(* CODESYS project raduga_prod.project

Project tree, tasks and I/O mapping:
  Device : Owen SPK2xx 03.CS.WEB, Owen, order no. 023, version 3.5.4.20
    application Application
      libraries: Standard, * (System); Util, 3.5.1.0 (System)
      task MainTask (cyclic, interval t#200ms, priority 2) calls PLC_PRG
      task VISU_TASK (cyclic, interval t#200ms, priority 30) calls VisuElems.Visu_Prg
      task AlarmManagerTask (cyclic, interval 50 ms, priority 31) calls AlarmManager.Alarm_Prg
      task bus_task (cyclic, interval t#100ms, priority 1, watchdog t#1000ms x 1) calls MV110
      program PLC_PRG [ST]
      visualisation Visualization
      Alarm Configuration
        alarm class Error (priority 10, acknowledge REP_ACK)
        alarm class Warning (priority 30, acknowledge REP)
        AlarmStorage
        text list AlarmGroup
        alarm group AlarmGroup
            3 [Error]: Comparison Equal, ExpressionToCompare TRUE, Expression PLC_PRG.alm_1 - "Ошибка_1"
            4 [Error]: Comparison Equal, ExpressionToCompare TRUE, Expression PLC_PRG.alm_2 - "Ошибка_2"
            6 [Warning]: Comparison Equal, ExpressionToCompare TRUE, Expression PLC_PRG.accident_sectional_machine - "Авария секционного автомата"
            7 [Warning]: Comparison Equal, ExpressionToCompare TRUE, Expression PLC_PRG.accident_input_1 - "Авария ввода №1"
            44 [Warning]: Comparison Equal, ExpressionToCompare FALSE, Expression PLC_PRG.accident_no_voltage_sec - "Отсутствует напряжение на секции"
            17 [Warning]: Comparison Greater, ExpressionToCompare 32, Expression PLC_PRG.module_in1_Ic - "Перегрузка Ic на вводе №1"
            15 [Warning]: Comparison Greater, ExpressionToCompare 32, Expression PLC_PRG.module_in1_Ia - "Перегрузка Ia на вводе №1"
            25 [Warning]: Comparison Greater, ExpressionToCompare 32, Expression PLC_PRG.module_in2_Ib - "Перегрузка Ib на вводе №2"
            35 [Warning]: Comparison Less, ExpressionToCompare 176, Expression PLC_PRG.module_v1_u3 - "Пониженное напряжение на секции №1 Uc = TRIGGERVALUE"
            13 [Warning]: Comparison Greater, ExpressionToCompare 264, Expression PLC_PRG.module_in1_u3 - "Повышенное напряжение на вводе №1 Uc = TRIGGERVALUE"
            23 [Warning]: Comparison Less, ExpressionToCompare 176, Expression PLC_PRG.module_in2_u3 - "Пониженное напряжение на вводе №2 Uc = TRIGGERVALUE"
            33 [Warning]: Comparison Less, ExpressionToCompare 176, Expression PLC_PRG.module_v1_u2 - "Пониженное напряжение на секции №1 Ub = TRIGGERVALUE"
            43 [Warning]: Comparison Equal, ExpressionToCompare FALSE, Expression PLC_PRG.accident_no_voltage_in_2 - "Отсутствует напряжение на вводе №2"
            21 [Warning]: Comparison Less, ExpressionToCompare 176, Expression PLC_PRG.module_in2_u2 - "Пониженное напряжение на вводе №2 Ub = TRIGGERVALUE"
            31 [Warning]: Comparison Less, ExpressionToCompare 176, Expression PLC_PRG.module_v1_u1 - "Пониженное напряжени на секции №1 Ua = TRIGGERVALUE"
            19 [Warning]: Comparison Less, ExpressionToCompare 176, Expression PLC_PRG.module_in2_u1 - "Пониженное напряжение  на вводе №2 Ua = TRIGGERVALUE"
            16 [Warning]: Comparison Greater, ExpressionToCompare 32, Expression PLC_PRG.module_in1_Ib - "Перегрузка Ib на вводе №1"
            26 [Warning]: Comparison Greater, ExpressionToCompare 32, Expression PLC_PRG.module_in2_Ic - "Перегрузка Ic на вводе №2"
            11 [Warning]: Comparison Greater, ExpressionToCompare 264, Expression PLC_PRG.module_in1_u2 - "Повышенное напряжение на вводе №1 Ub = TRIGGERVALUE"
            14 [Warning]: Comparison Less, ExpressionToCompare 176, Expression PLC_PRG.module_in1_u3 - "Пониженное напряжение Uc на вводе №1 = TRIGGERVALUE"
            24 [Warning]: Comparison Greater, ExpressionToCompare 32, Expression PLC_PRG.module_in2_Ia - "Перегрузка Ia на вводе №2"
            34 [Warning]: Comparison Greater, ExpressionToCompare 264, Expression PLC_PRG.module_v1_u3 - "Повышенное напряжение на секции №1 Uc = TRIGGERVALUE"
            12 [Warning]: Comparison Less, ExpressionToCompare 176, Expression PLC_PRG.module_in1_u2 - "Пониженное напряжение на вводе №1 Ub = TRIGGERVALUE"
            22 [Warning]: Comparison Greater, ExpressionToCompare 264, Expression PLC_PRG.module_in2_u3 - "Повышенное напряжение на вводе №2 Uc = TRIGGERVALUE"
            32 [Warning]: Comparison Greater, ExpressionToCompare 264, Expression PLC_PRG.module_v1_u2 - "Повышенное напряжение на секции №1 Ub = TRIGGERVALUE"
            10 [Warning]: Comparison Less, ExpressionToCompare 176, Expression PLC_PRG.module_in1_u1 - "Пониженное напряжение  на вводе №1 Ua = TRIGGERVALUE"
            20 [Warning]: Comparison Greater, ExpressionToCompare 264, Expression PLC_PRG.module_in2_u2 - "Повышенное напряжение на вводе №2 Ub = TRIGGERVALUE "
            30 [Warning]: Comparison Greater, ExpressionToCompare 264, Expression PLC_PRG.module_v1_u1 - "Повышенное напряжение на секции №1 Ua = TRIGGERVALUE"
            42 [Warning]: Comparison Equal, ExpressionToCompare FALSE, Expression PLC_PRG.accident_no_voltage_in_1 - "Отсутствует напряжение на вводе №1"
            18 [Warning]: Comparison Greater, ExpressionToCompare 264, Expression PLC_PRG.module_in2_u1 - "Повышенное напряжение  на вводе №2 Ua = TRIGGERVALUE"
            8 [Warning]: Comparison Equal, ExpressionToCompare TRUE, Expression PLC_PRG.accident_input_2 - "Авария ввода №2"
            9 [Warning]: Comparison Greater, ExpressionToCompare 264, Expression PLC_PRG.module_in1_u1 - "Повышенное напряжение  на вводе №1 Ua = TRIGGERVALUE"
            0 [Warning]: Comparison Equal, ExpressionToCompare TRUE, Expression PLC_PRG.war_1 - "Предупреждение_1"
            1 [Warning]: Comparison Equal, ExpressionToCompare TRUE, Expression PLC_PRG.war_2 - "Предупреждение_2"
      function block Two_words_to_Real [ST]
      visualisation volt_1
      visualisation mpx_1
      visualisation mpx_2
      visualisation scheme
      image pool ImagePool
    Modbus_COM : Modbus COM, 3S - Smart Software Solutions GmbH, version 3.4.0.0
        settings: DataBits = 8; StopBits = 1; ComPort = 3
      Modbus_Master_COM_Port : Modbus Master, COM Port, 3S - Smart Software Solutions GmbH, version 3.5.5.0
          settings: Transmission = 'RTU'; ResponseTimeout = 1000; TimeBetweenFrames = 10; Auto-restart communication = TRUE
        MV110 : Modbus Slave, COM Port, 3S - Smart Software Solutions GmbH, version 3.5.4.0
            settings: SlaveAddress = 10; ResponseTimeout = 1000; UseExtendedFunctionCodes = TRUE; Channel 0.Function Code = 3; Channel 0.Read Offset = 16#0033; Channel 0.Read Length = 1; Channel 0.Write Offset = 0; Channel 0.Write Length = 0; Channel 0.Cycle Time = 500
            input  Application.PLC_PRG.module_mv110_reg1 : WORD  // Channel 0.Channel 0
            unmapped channels: Channel 0
        MPX_1 : Modbus Slave, COM Port, 3S - Smart Software Solutions GmbH, version 3.5.4.0
            settings: SlaveAddress = 11; ResponseTimeout = 1000; UseExtendedFunctionCodes = TRUE; Input_group.Function Code = 4; Input_group.Read Offset = 16#000B; Input_group.Read Length = 7; Input_group.Write Offset = 0; Input_group.Write Length = 0; Input_group.Cycle Time = 500; Bypass_out_group.Function Code = 3; Bypass_out_group.Read Offset = 16#0015; Bypass_out_group.Read Length = 7; Bypass_out_group.Write Offset = 0; Bypass_out_group.Write Length = 0; Bypass_out_group.Cycle Time = 500; Output_group.Function Code = 3; Output_group.Read Offset = 16#001F; Output_group.Read Length = 13; Output_group.Write Offset = 0; Output_group.Write Length = 0; Output_group.Cycle Time = 500; Battery_group.Function Code = 3; Battery_group.Read Offset = 16#002F; Battery_group.Read Length = 7; Battery_group.Write Offset = 0; Battery_group.Write Length = 0; Battery_group.Cycle Time = 500; temp.Function Code = 3; temp.Read Offset = 16#003D; temp.Read Length = 1; temp.Write Offset = 0; temp.Write Length = 0; temp.Cycle Time = 500; states.Function Code = 3; states.Read Offset = 16#0000; states.Read Length = 2; states.Write Offset = 0; states.Write Length = 0; states.Cycle Time = 500
            input  Application.PLC_PRG.mpx1_in_v_1 : WORD  // Input_group.Input_group
            input  Application.PLC_PRG.mpx1_in_v_2 : WORD  // Input_group.Input_group
            input  Application.PLC_PRG.mpx1_in_v_3 : WORD  // Input_group.Input_group
            input  Application.PLC_PRG.mpx1_in_i_1 : WORD  // Input_group.Input_group
            input  Application.PLC_PRG.mpx1_in_i_2 : WORD  // Input_group.Input_group
            input  Application.PLC_PRG.mpx1_in_i_3 : WORD  // Input_group.Input_group
            input  Application.PLC_PRG.mpx1_in_freq : WORD  // Input_group.Input_group
            input  Application.PLC_PRG.mpx1_bypass_v_1 : WORD  // Bypass_out_group.Bypass_out_group
            input  Application.PLC_PRG.mpx1_bypass_v_2 : WORD  // Bypass_out_group.Bypass_out_group
            input  Application.PLC_PRG.mpx1_bypass_v_3 : WORD  // Bypass_out_group.Bypass_out_group
            input  Application.PLC_PRG.mpx1_bypass_freq : WORD  // Bypass_out_group.Bypass_out_group
            input  Application.PLC_PRG.mpx1_output_v_1 : WORD  // Bypass_out_group.Bypass_out_group
            input  Application.PLC_PRG.mpx1_output_v_2 : WORD  // Bypass_out_group.Bypass_out_group
            input  Application.PLC_PRG.mpx1_output_v_3 : WORD  // Bypass_out_group.Bypass_out_group
            input  Application.PLC_PRG.mpx1_output_i_1 : WORD  // Output_group.Output_group
            input  Application.PLC_PRG.mpx1_output_i_2 : WORD  // Output_group.Output_group
            input  Application.PLC_PRG.mpx1_output_i_3 : WORD  // Output_group.Output_group
            input  Application.PLC_PRG.mpx1_load_ph_1 : WORD  // Output_group.Output_group
            input  Application.PLC_PRG.mpx1_load_ph_2 : WORD  // Output_group.Output_group
            input  Application.PLC_PRG.mpx1_load_ph_3 : WORD  // Output_group.Output_group
            input  Application.PLC_PRG.mpx1_output_active_power_1 : WORD  // Output_group.Output_group
            input  Application.PLC_PRG.mpx1_output_active_power_2 : WORD  // Output_group.Output_group
            input  Application.PLC_PRG.mpx1_output_active_power_3 : WORD  // Output_group.Output_group
            input  Application.PLC_PRG.mpx1_output_freq : WORD  // Output_group.Output_group
            input  Application.PLC_PRG.mpx1_battery_voltage : WORD  // Battery_group.Battery_group
            input  Application.PLC_PRG.mpx1_battery_current : WORD  // Battery_group.Battery_group
            input  Application.PLC_PRG.mpx1_battery_capacity : WORD  // Battery_group.Battery_group
            input  Application.PLC_PRG.mpx1_battery_time : WORD  // Battery_group.Battery_group
            input  Application.PLC_PRG.mpx1_temp : WORD  // temp.temp
            input  Application.PLC_PRG.mpx1_state_reg_1 : WORD  // states.states
            input  Application.PLC_PRG.mpx1_state_reg_2 : WORD  // states.states
            unmapped channels: Input_group, Bypass_out_group, Output_group, Battery_group, temp, states
    Modbus_slave : Modbus COM, 3S - Smart Software Solutions GmbH, version 3.4.0.0
        settings: DataBits = 8; StopBits = 1; ComPort = 4
      Modbus_Serial_Device : Modbus Serial Device, 3S - Smart Software Solutions GmbH, version 3.5.3.80
          settings: Unit-ID = 3
          unmapped channels: Inputs, Outputs
    Ethernet : Ethernet, 3S - Smart Software Solutions GmbH, version 3.4.2.0
      Modbus_TCP_Master : Modbus TCP Master, 3S - Smart Software Solutions GmbH, version 3.5.4.0
          settings: AutoReconnect = TRUE
        IPS_1 : Modbus TCP Slave, 3S - Smart Software Solutions GmbH, version 3.5.4.0
            settings: Unit-ID = 1; ResponseTimeout = 1500; IPAddress = [192, 168, 19, 34]; Input_group.Function Code = 3; Input_group.Read Offset = 16#006E; Input_group.Read Length = 3; Input_group.Write Offset = 0; Input_group.Write Length = 0; Input_group.Cycle Time = 500; Output_group.Function Code = 3; Output_group.Read Offset = 16#0077; Output_group.Read Length = 7; Output_group.Write Offset = 0; Output_group.Write Length = 0; Output_group.Cycle Time = 500; Bypass_group.Function Code = 3; Bypass_group.Read Offset = 16#0081; Bypass_group.Read Length = 4; Bypass_group.Write Offset = 0; Bypass_group.Write Length = 0; Bypass_group.Cycle Time = 500
            unmapped channels: Input_group, Output_group, Bypass_group
    Modbus_PLC_slave : Modbus COM, 3S - Smart Software Solutions GmbH, version 3.4.0.0
        settings: DataBits = 8; StopBits = 1; ComPort = 2
      Modbus_Serial_Device_1 : Modbus Serial Device, 3S - Smart Software Solutions GmbH, version 3.5.5.0
          unmapped channels: Inputs, Outputs
  text list GlobalTextList
  5ce3da45-db07-42e7-a21c-a00fff4ed8f6|D:\scheme_3.png
  5ce3da45-db07-42e7-a21c-a00fff4ed8f6|D:\scheme.png
  5ce3da45-db07-42e7-a21c-a00fff4ed8f6|D:\on.png
  5ce3da45-db07-42e7-a21c-a00fff4ed8f6|D:\off.png
  5ce3da45-db07-42e7-a21c-a00fff4ed8f6|D:\off.jpg
  5ce3da45-db07-42e7-a21c-a00fff4ed8f6|D:\on.jpg
  5ce3da45-db07-42e7-a21c-a00fff4ed8f6|D:\on_ind.jpg
  5ce3da45-db07-42e7-a21c-a00fff4ed8f6|D:\off_ind.jpg
  5ce3da45-db07-42e7-a21c-a00fff4ed8f6|D:\entel.png
  5ce3da45-db07-42e7-a21c-a00fff4ed8f6|D:\zit.png
  5ce3da45-db07-42e7-a21c-a00fff4ed8f6|D:\entel.jpg
  5ce3da45-db07-42e7-a21c-a00fff4ed8f6|D:\zit.jpg
  5ce3da45-db07-42e7-a21c-a00fff4ed8f6|D:\vvod_off.png
  5ce3da45-db07-42e7-a21c-a00fff4ed8f6|D:\vvod_on.png
*)

// Device/Application/PLC_PRG
PROGRAM PLC_PRG
VAR
	alm_1: BOOL;
	alm_2: BOOL;
	war_1: BOOL;
	war_2: BOOL;
	//Переменные для отработки аварийных ситуаций
	accident_sectional_machine :BOOL := FALSE; //авария секционного автомата
	accident_input_1		   :BOOL := FALSE; //авария ввода №1
	accident_input_2		   :BOOL := FALSE; //авария ввода №2
	accident_no_voltage_in_1   :BOOL := FALSE; //отсутствие напряжения на вводе №1
	accident_no_voltage_in_2   :BOOL := FALSE; //отсутствие напряжения на вводе №2
	manual_mode				   :BOOL := FALSE;
	auto_mode                  :BOOL := FALSE;
	remote_mode                :BOOL := FALSE;
	accident_no_voltage_sec    :BOOL := FALSE; //отсутствие напряжения на секции
	
	ack:BOOL;
	history:BOOL;
	
	//Переменные для работы с MPX_1
	mpx1_in_v_1 	 		:WORD; //1-е Напрядение входа
	mpx1_in_v_2 	 :WORD; //2-e Напряжение входа
	mpx1_in_v_3 	 :WORD; //3-е Напряжение входа
	mpx1_in_i_1 	 :WORD; //1-й Ток входа
	mpx1_in_i_2 	 :WORD; //2-й Ток входа
	mpx1_in_i_3 	 :WORD; //3-й Ток входа
	mpx1_in_freq 	 :WORD; //Частота на входе
	mpx1_bypass_v_1  :WORD; //1-е Напряжение байпаса
	mpx1_bypass_v_2  :WORD; //2-е Напряжение байпаса
	mpx1_bypass_v_3  :WORD; //3-е Напряжение байпаса
	mpx1_bypass_freq :WORD; //Частота байпаса
	mpx1_output_v_1  :WORD; //1-е Напряжение выхода
	mpx1_output_v_2  :WORD; //2-е Напряжение выхода
	mpx1_output_v_3  :WORD; //3-е Напряжение выхода
	mpx1_output_i_1  :WORD; //1-й Ток выхода
	mpx1_output_i_2  		   :WORD; //2-й Ток выхода
	mpx1_output_i_3  		   :WORD; //3-й Ток выхода
	mpx1_output_active_power_1 :WORD; //Активная мощность 1-й фазы
	mpx1_output_active_power_2 :WORD; //Активная мощность 2-й фазы
	mpx1_output_active_power_3 :WORD; //Активная мощность 3-й фазы
	mpx1_output_freq :WORD; //Частота выхода
	mpx1_load_ph_1    :WORD; //Загрузска 1-й фазы (%)
	mpx1_load_ph_2    :WORD; //Загрузска 3-й фазы (%)
	mpx1_load_ph_3    :WORD; //Загрузска 2-й фазы (%)
	mpx1_battery_voltage :WORD; //Напряжение батареи
	mpx1_battery_current :WORD; //Ток батареи
	mpx1_battery_capacity :WORD; //Остаточная емкость батареи (%)
	mpx1_battery_time :WORD; //Остаточное время автономии (минуты)
	mpx1_temp :WORD; //Температура
	mpx1_state_reg_1 :WORD; //1-й Регистр состояния
	mpx1_state_1_as_bit :WORD_AS_BIT;
	mpx1_state_reg_2 :WORD; //2-й Регистр состояния
	mpx1_state_2_as_bit :WORD_AS_BIT;
	
	
	
	//Переменные для работы с первым МВ110-16 (адрес = 1)
	module_mv110_reg1	:WORD; //Первый регистр состояния входов МВ110-16
	mv110_reg_as_bit 	:WORD_AS_BIT; 
	mv110_in_1 			:STRING; //РКН ввода 1
	mv110_in_2 			:STRING; //РКН ввода 2
	mv110_in_3 			:STRING; //Сборная шина 1
	mv110_in_4 			:STRING; //Сборная шина 2
	mv110_in_5 			:STRING; //Авария секционного автомата
	mv110_in_6 			:STRING; //Авария ввода 1
	mv110_in_7 			:STRING; //Авария ввода 2
	mv110_in_9 			:STRING; //Положение секционного авт.
	mv110_in_10			:STRING; //Положение ввода 1 авт.
	mv110_in_11			:STRING; //Положение ввода 2 авт.
	mode                :WSTRING := "Старт"; //Режим работы (ручной, ручной дистанционный, автоматический)
	
	
	//Переменные для работы с первым вольтметром (адрес = 3)
	module_v1_u1		:REAL; //Значение Ua первого вольтметра
	module_v1_u2		:REAL; //Значение Ub первого вольтметра
	module_v1_u3		:REAL; //Значение Uc первого вольтметра	
	module_v1_u1_reg1	:WORD; //Первый регистр Ua первого вольтметра
	module_v1_u1_reg2	:WORD; //Второй регистр Ua первого вольтметра
	module_v1_u2_reg1	:WORD; //Первый регистр Ub первого вольтметра
	module_v1_u2_reg2	:WORD; //Второй регистр Ub первого вольтметра
	module_v1_u3_reg1	:WORD; //Первый регистр Uс первого вольтметра
	module_v1_u3_reg2	:WORD; //Второй регистр Uс первого вольтметра		
	module_v1_u1_convertion: Two_words_to_Real;
	module_v1_u2_convertion: Two_words_to_Real;
	module_v1_u3_convertion: Two_words_to_Real;	
	module_v1_F			:REAL; //Значение частоты первого вольтметра	
	module_v1_F_reg1	:WORD; //Первый регистр F первого вольтметра
	module_v1_F_reg2	:WORD; //Второй регистр F первого вольтметра	
	module_v1_F_convertion: Two_words_to_Real;
		
	//Переменные для работы с первым вводом (адрес = 5)
	module_in1_u1		:REAL; //Значение Ua первого ввода
	module_in1_u2		:REAL; //Значение Ub первого ввода
	module_in1_u3		:REAL; //Значение Uc первого ввода	
	module_in1_u1_reg1	:WORD; //Первый регистр Ua первого ввода
	module_in1_u1_reg2	:WORD; //Второй регистр Ua первого ввода
	module_in1_u2_reg1	:WORD; //Первый регистр Ub первого ввода
	module_in1_u2_reg2	:WORD; //Второй регистр Ub первого ввода
	module_in1_u3_reg1	:WORD; //Первый регистр Uс первого ввода
	module_in1_u3_reg2	:WORD; //Второй регистр Uс первого ввода		
	module_in1_u1_convertion: Two_words_to_Real;
	module_in1_u2_convertion: Two_words_to_Real;
	module_in1_u3_convertion: Two_words_to_Real;
	
	module_in1_Uab		:REAL; //Значение Uab первого ввода
	module_in1_Ubc		:REAL; //Значение Ubc первого ввода
	module_in1_Uca		:REAL; //Значение Uca первого ввода	
	module_in1_Uab_reg1	:WORD; //Первый регистр Uab первого ввода
	module_in1_Uab_reg2	:WORD; //Второй регистр Uab первого ввода
	module_in1_Ubc_reg1	:WORD; //Первый регистр Ubc первого ввода
	module_in1_Ubc_reg2	:WORD; //Второй регистр Ubc первого ввода
	module_in1_Uca_reg1	:WORD; //Первый регистр Uсa первого ввода
	module_in1_Uca_reg2	:WORD; //Второй регистр Uсa первого ввода	
	module_in1_Uab_convertion: Two_words_to_Real;
	module_in1_Ubc_convertion: Two_words_to_Real;
	module_in1_Uca_convertion: Two_words_to_Real;
	
	module_in1_Ia		:REAL; //Значение Ia первого ввода
	module_in1_Ib		:REAL; //Значение Ib первого ввода
	module_in1_Ic		:REAL; //Значение Ic первого ввода	
	module_in1_Ia_reg1	:WORD; //Первый регистр Ia первого ввода
	module_in1_Ia_reg2	:WORD; //Второй регистр Ia первого ввода
	module_in1_Ib_reg1	:WORD; //Первый регистр Ib первого ввода
	module_in1_Ib_reg2	:WORD; //Второй регистр Ib первого ввода
	module_in1_Ic_reg1	:WORD; //Первый регистр Iс первого ввода
	module_in1_Ic_reg2	:WORD; //Второй регистр Iс первого ввода	
	module_in1_Ia_convertion: Two_words_to_Real;
	module_in1_Ib_convertion: Two_words_to_Real;
	module_in1_Ic_convertion: Two_words_to_Real;

	module_in1_F		:REAL; //Значение частоты первого ввода
	module_in1_F_reg1	:WORD; //Первый регистр F первого ввода
	module_in1_F_reg2	:WORD; //Второй регистр F первого ввода	
	module_in1_F_convertion: Two_words_to_Real;
	
	//Переменные для работы со вторым вводом (адрес = 6)
	module_in2_u1		:REAL; //Значение Ua первого второго
	module_in2_u2		:REAL; //Значение Ub первого второго
	module_in2_u3		:REAL; //Значение Uc первого второго	
	module_in2_u1_reg1	:WORD; //Первый регистр Ua первого второго
	module_in2_u1_reg2	:WORD; //Второй регистр Ua первого второго
	module_in2_u2_reg1	:WORD; //Первый регистр Ub первого второго
	module_in2_u2_reg2	:WORD; //Второй регистр Ub первого второго
	module_in2_u3_reg1	:WORD; //Первый регистр Uс первого второго
	module_in2_u3_reg2	:WORD; //Второй регистр Uс первого второго		
	module_in2_u1_convertion: Two_words_to_Real;
	module_in2_u2_convertion: Two_words_to_Real;
	module_in2_u3_convertion: Two_words_to_Real;
	
	module_in2_Uab		:REAL; //Значение Uab первого ввода
	module_in2_Ubc		:REAL; //Значение Ubc первого ввода
	module_in2_Uca		:REAL; //Значение Uca первого ввода	
	module_in2_Uab_reg1	:WORD; //Первый регистр Uab первого ввода
	module_in2_Uab_reg2	:WORD; //Второй регистр Uab первого ввода
	module_in2_Ubc_reg1	:WORD; //Первый регистр Ubc первого ввода
	module_in2_Ubc_reg2	:WORD; //Второй регистр Ubc первого ввода
	module_in2_Uca_reg1	:WORD; //Первый регистр Uсa первого ввода
	module_in2_Uca_reg2	:WORD; //Второй регистр Uсa первого ввода	
	module_in2_Uab_convertion: Two_words_to_Real;
	module_in2_Ubc_convertion: Two_words_to_Real;
	module_in2_Uca_convertion: Two_words_to_Real;

	module_in2_Ia		:REAL; //Значение Ia первого ввода
	module_in2_Ib		:REAL; //Значение Ib первого ввода
	module_in2_Ic		:REAL; //Значение Ic первого ввода	
	module_in2_Ia_reg1	:WORD; //Первый регистр Ia первого ввода
	module_in2_Ia_reg2	:WORD; //Второй регистр Ia первого ввода
	module_in2_Ib_reg1	:WORD; //Первый регистр Ib первого ввода
	module_in2_Ib_reg2	:WORD; //Второй регистр Ib первого ввода
	module_in2_Ic_reg1	:WORD; //Первый регистр Iс первого ввода
	module_in2_Ic_reg2	:WORD; //Второй регистр Iс первого ввода	
	module_in2_Ia_convertion: Two_words_to_Real;
	module_in2_Ib_convertion: Two_words_to_Real;
	module_in2_Ic_convertion: Two_words_to_Real;
	
	module_in2_F		:REAL; //Значение частоты первого ввода
	module_in2_F_reg1	:WORD; //Первый регистр F первого ввода
	module_in2_F_reg2	:WORD; //Второй регистр F первого ввода	
	module_in2_F_convertion: Two_words_to_Real;
END_VAR

//Конвертация параметров mpx_1




//Конвертация 2 считанных регистров типа WORD в одну переменную REAL для каждого измеряемого значения
//Первый вольтметр (адрес = 3)
module_v1_u1_convertion(Inpit_1:=module_v1_u1_reg1 , Inpit_2:=module_v1_u1_reg2 , output=>module_v1_u1 ); //V1 Ua
module_v1_u2_convertion(Inpit_1:=module_v1_u2_reg1 , Inpit_2:=module_v1_u2_reg2 , output=>module_v1_u2 ); //V1 Ub
module_v1_u3_convertion(Inpit_1:=module_v1_u3_reg1 , Inpit_2:=module_v1_u3_reg2 , output=>module_v1_u3 ); //V1 Uc
module_v1_F_convertion  (Inpit_1:=module_v1_F_reg1,    Inpit_2 := module_v1_F_reg2,   output=>module_v1_F );   //V1 F

//МФИ ввод №1 (адрес = 5)
module_in1_u1_convertion(Inpit_1:=module_in1_u1_reg1 , Inpit_2:=module_in1_u1_reg2 , output=>module_in1_u1 ); //Ua
module_in1_u2_convertion(Inpit_1:=module_in1_u2_reg1 , Inpit_2:=module_in1_u2_reg2 , output=>module_in1_u2 ); //Ub
module_in1_u3_convertion(Inpit_1:=module_in1_u3_reg1 , Inpit_2:=module_in1_u3_reg2 , output=>module_in1_u3 ); //Uc
module_in1_Uab_convertion(Inpit_1:=module_in1_Uab_reg1,  Inpit_2 := module_in1_Uab_reg2, output=>module_in1_Uab ); //Uab
module_in1_Ubc_convertion(Inpit_1:=module_in1_Ubc_reg1,  Inpit_2 := module_in1_Ubc_reg2, output=>module_in1_Ubc ); //Ubc
module_in1_Uca_convertion(Inpit_1:=module_in1_Uca_reg1,  Inpit_2 := module_in1_Uca_reg2, output=>module_in1_Uca ); //Uca
module_in1_F_convertion  (Inpit_1:=module_in1_F_reg1,    Inpit_2 := module_in1_F_reg2,   output=>module_in1_F );//F
module_in1_Ia_convertion  (Inpit_1:=module_in1_Ia_reg1,    Inpit_2 := module_in1_Ia_reg2,   output=>module_in1_Ia );//Ia
module_in1_Ib_convertion  (Inpit_1:=module_in1_Ib_reg1,    Inpit_2 := module_in1_Ib_reg2,   output=>module_in1_Ib );//Ib
module_in1_Ic_convertion  (Inpit_1:=module_in1_Ic_reg1,    Inpit_2 := module_in1_Ic_reg2,   output=>module_in1_Ic );//Ic

//МФИ ввод №2 (адрес = 6)
module_in2_u1_convertion(Inpit_1:=module_in2_u1_reg1 , Inpit_2:=module_in2_u1_reg2 , output=>module_in2_u1 ); //Ua
module_in2_u2_convertion(Inpit_1:=module_in2_u2_reg1 , Inpit_2:=module_in2_u2_reg2 , output=>module_in2_u2 ); //Ub
module_in2_u3_convertion(Inpit_1:=module_in2_u3_reg1 , Inpit_2:=module_in2_u3_reg2 , output=>module_in2_u3 ); //Uc
module_in2_Uab_convertion(Inpit_1:=module_in2_Uab_reg1,  Inpit_2 := module_in2_Uab_reg2, output=>module_in2_Uab ); //Uab
module_in2_Ubc_convertion(Inpit_1:=module_in2_Ubc_reg1,  Inpit_2 := module_in2_Ubc_reg2, output=>module_in2_Ubc ); //Ubc
module_in2_Uca_convertion(Inpit_1:=module_in2_Uca_reg1,  Inpit_2 := module_in2_Uca_reg2, output=>module_in2_Uca ); //Uca
module_in2_F_convertion  (Inpit_1:=module_in2_F_reg1,    Inpit_2 := module_in2_F_reg2,   output=>module_in2_F );//F
module_in2_Ia_convertion  (Inpit_1:=module_in2_Ia_reg1,    Inpit_2 := module_in2_Ia_reg2,   output=>module_in2_Ia );//Ia
module_in2_Ib_convertion  (Inpit_1:=module_in2_Ib_reg1,    Inpit_2 := module_in2_Ib_reg2,   output=>module_in2_Ib );//Ib
module_in2_Ic_convertion  (Inpit_1:=module_in2_Ic_reg1,    Inpit_2 := module_in2_Ic_reg2,   output=>module_in2_Ic );//Ic

//Логика МВ110-16
mv110_reg_as_bit(W := module_mv110_reg1);

IF (mv110_reg_as_bit.B00 = FALSE) THEN
	mv110_in_1 := 'on_ind';
	ELSE
		mv110_in_1 := 'off_ind';	
END_IF
IF (mv110_reg_as_bit.B01 = FALSE) THEN
	mv110_in_2 := 'on_ind';
	ELSE
		mv110_in_2 := 'off_ind';	 
END_IF
IF (mv110_reg_as_bit.B02 = FALSE) THEN
	mv110_in_3 := 'on_ind';
	ELSE
		mv110_in_3 := 'off_ind';	 
END_IF
IF (mv110_reg_as_bit.B03 = FALSE) THEN
	mv110_in_4 := 'on_ind';
	ELSE
		mv110_in_4 := 'off_ind';	 
END_IF
IF (mv110_reg_as_bit.B08 = TRUE) THEN
	mv110_in_9 := 'on';
	ELSE
		mv110_in_9 := 'off';	 
END_IF
IF (mv110_reg_as_bit.B09 = TRUE) THEN
	mv110_in_10 := 'on';
	ELSE
		mv110_in_10 := 'off';	 
END_IF
IF (mv110_reg_as_bit.B10 = TRUE) THEN
	mv110_in_11 := 'on';
	ELSE
		mv110_in_11 := 'off';	 	 
END_IF
IF (mv110_reg_as_bit.B04 = TRUE) THEN
	accident_sectional_machine := TRUE;
	ELSE
		accident_sectional_machine := FALSE;	 	 
END_IF
IF (mv110_reg_as_bit.B05 = TRUE) THEN
	accident_input_1 := TRUE;
	ELSE
		accident_input_1 := FALSE;	 	 
END_IF
IF (mv110_reg_as_bit.B06 = TRUE) THEN
	accident_input_2 := TRUE;
	ELSE
		accident_input_2 := FALSE;	 	 
END_IF
IF (mv110_reg_as_bit.B00 = FALSE) THEN
	accident_no_voltage_in_1 := FALSE;
	ELSE
		accident_no_voltage_in_1 := TRUE;	
END_IF
IF (mv110_reg_as_bit.B01 = FALSE) THEN
	accident_no_voltage_in_2 := FALSE;
	ELSE
		accident_no_voltage_in_2 := TRUE;	 
END_IF
IF (mv110_reg_as_bit.B02 = FALSE) THEN
	accident_no_voltage_sec := FALSE;
	ELSE
		accident_no_voltage_sec := TRUE;	 
END_IF
IF (mv110_reg_as_bit.B12 = TRUE) THEN
	mode := "Автоматический";
	auto_mode := TRUE;
	manual_mode := FALSE;
	remote_mode := FALSE;
END_IF
IF ((mv110_reg_as_bit.B12 = FALSE) AND (mv110_reg_as_bit.B13 = FALSE)) THEN
	mode := "Ручной";
	auto_mode := FALSE;
	manual_mode := TRUE;
	remote_mode := FALSE;
END_IF
IF ((mv110_reg_as_bit.B12 = FALSE) AND (mv110_reg_as_bit.B13 = TRUE)) THEN
	mode := "Дистанционный";
	auto_mode := FALSE;
	manual_mode := FALSE;
	remote_mode := TRUE;
END_IF
//--------------------------


(*открыли порт 3. я откатил до старых версий порты , компилируется.
добавил чтение раз в 100 мс регистра 2и 3 в канале нуль
в закладке соотнесение указал включено 2 = для обновления данных в СПК циклично
склейл два ворда в реал в первой строке этого кода
далее код переподъём  ,в случае  ,если модуль упал ( убрали или ошибки)*)

END_PROGRAM

// Device/Application/Two_words_to_Real
FUNCTION_BLOCK Two_words_to_Real
VAR_INPUT
	Inpit_1:WORD;
	Inpit_2:WORD;
END_VAR
VAR_OUTPUT
	output:real;
END_VAR
VAR
	P:POINTER TO ARRAY [0..3] OF BYTE; 
	pi1:POINTER TO ARRAY [0..1] OF BYTE; 
	pi2:POINTER TO ARRAY [0..1] OF BYTE; 
END_VAR

pi1:=ADR(Inpit_1);
pi2:=ADR(Inpit_2);



P:=ADR(output);
P^[0]:=pi2^[0];
P^[1]:=pi2^[1];
P^[2]:=pi1^[0];
P^[3]:=pi1^[1];

END_FUNCTION_BLOCK

// Device/Application/Visualization
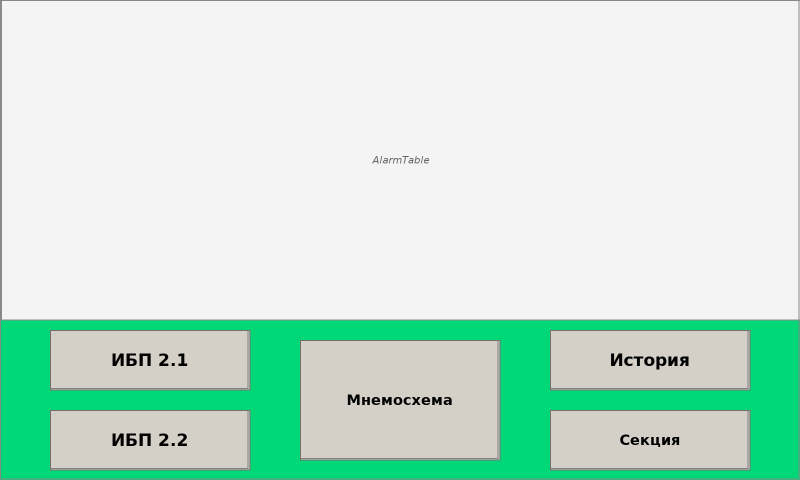
VISUALIZATION Visualization  // 800x480
    AlarmTable (1,0 800x320)
        Column[0]: ColumnTitle=Время
        Column[1]: ColumnTitle=Сообщение
        p1521930926: __All
        p1663851261: __All
        p428520879: PLC_PRG.ack
        p3266827225: PLC_PRG.history
    Button (550,330 200x60), "История", colour toggle: PLC_PRG.history
        toggle PLC_PRG.history
    Button (550,410 200x60), "Секция"
        OnMouseClick:  Assign=volt_1, Type=Assignment
    Button (50,330 200x60), "ИБП 2.1"
        OnMouseClick:  Assign=mpx_1, Type=Assignment
    Button (50,410 200x60), "ИБП 2.2"
        OnMouseClick:  Assign=mpx_2, Type=Assignment
    Button (300,340 200x120), "Мнемосхема"
        OnMouseClick:  Assign=scheme, Type=Assignment
END_VISUALIZATION

// Device/Application/volt_1
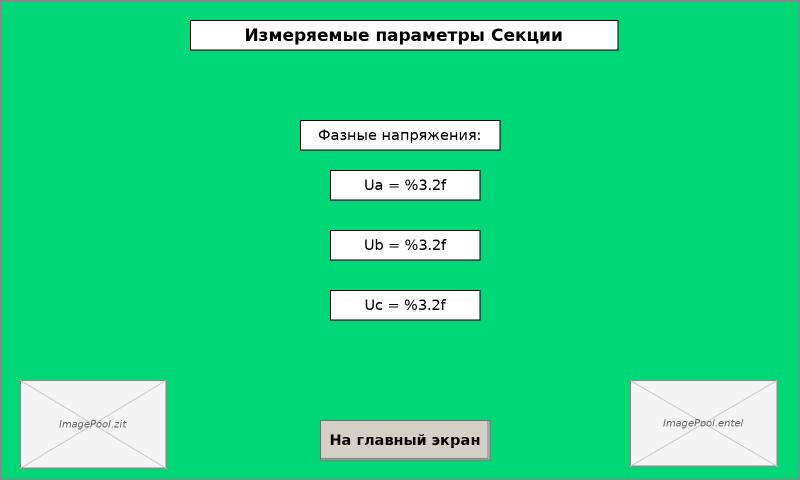
VISUALIZATION volt_1  // 800x480
    Rectangle (190,20 428x30), "Измеряемые параметры Секции"
    Button (320,420 170x40), "На главный экран"
        OnMouseClick:  Assign=Visualization, Type=Assignment
    Rectangle (300,120 200x30), "Фазные напряжения:"
    Rectangle (330,170 150x30), "Ua = %3.2f", text variable: PLC_PRG.module_v1_u1
    Rectangle (330,230 150x30), "Ub = %3.2f", text variable: PLC_PRG.module_v1_u2
    Rectangle (330,290 150x30), "Uc = %3.2f", text variable: PLC_PRG.module_v1_u3
    Image (630,380 147x86), image: ImagePool.entel
    Image (20,380 146x88), image: ImagePool.zit
END_VISUALIZATION

// Device/Application/mpx_1
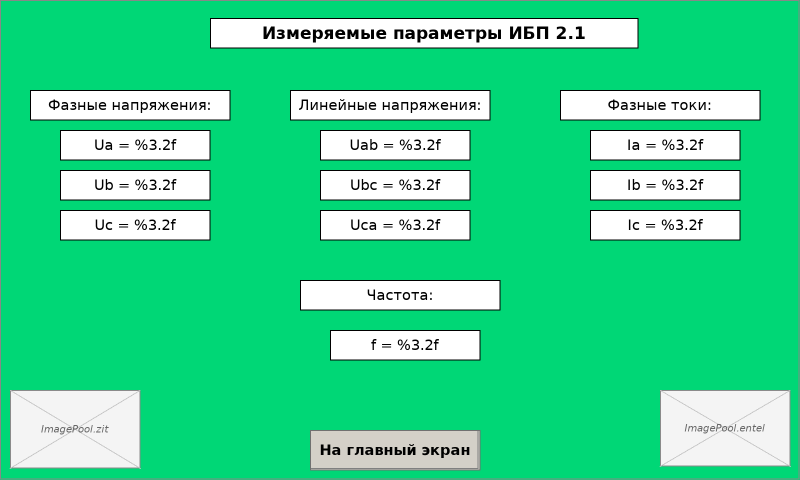
VISUALIZATION mpx_1  // 800x480
    Button (310,430 170x40), "На главный экран"
        OnMouseClick:  Assign=Visualization, Type=Assignment
    Rectangle (210,18 428x30), "Измеряемые параметры ИБП 2.1"
    Rectangle (30,90 200x30), "Фазные напряжения:"
    Rectangle (60,130 150x30), "Ua = %3.2f", text variable: PLC_PRG.module_in1_u1
    Rectangle (60,170 150x30), "Ub = %3.2f", text variable: PLC_PRG.module_in1_u2
    Rectangle (60,210 150x30), "Uc = %3.2f", text variable: PLC_PRG.module_in1_u3
    Rectangle (290,90 200x30), "Линейные напряжения:"
    Rectangle (320,130 150x30), "Uab = %3.2f", text variable: PLC_PRG.module_in1_Uab
    Rectangle (320,170 150x30), "Ubc = %3.2f", text variable: PLC_PRG.module_in1_Ubc
    Rectangle (320,210 150x30), "Uca = %3.2f", text variable: PLC_PRG.module_in1_Uca
    Rectangle (560,90 200x30), "Фазные токи:"
    Rectangle (590,130 150x30), "Ia = %3.2f", text variable: PLC_PRG.module_in1_Ia
    Rectangle (590,170 150x30), "Ib = %3.2f", text variable: PLC_PRG.module_in1_Ib
    Rectangle (590,210 150x30), "Ic = %3.2f", text variable: PLC_PRG.module_in1_Ic
    Rectangle (300,280 200x30), "Частота:"
    Rectangle (330,330 150x30), "f = %3.2f", text variable: PLC_PRG.module_in1_F
    Image (10,390 130x78), image: ImagePool.zit
    Image (660,390 130x76), image: ImagePool.entel
END_VISUALIZATION

// Device/Application/mpx_2
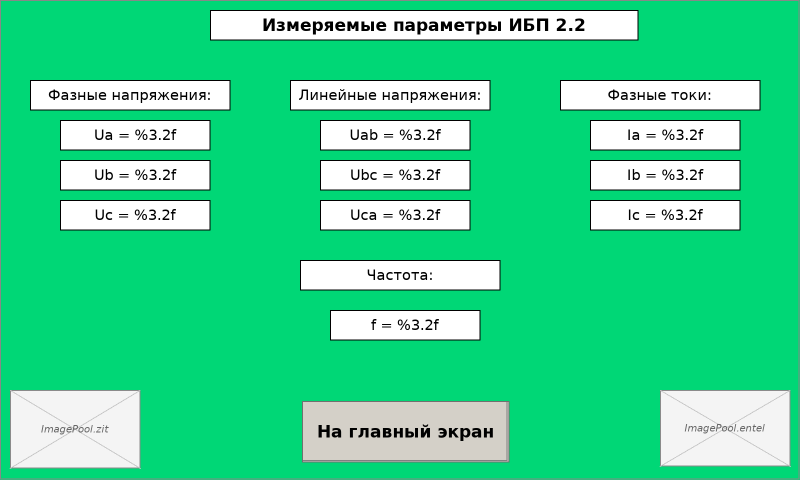
VISUALIZATION mpx_2  // 800x480
    Button (302,401 207x61), "На главный экран"
        OnMouseClick:  Assign=Visualization, Type=Assignment
    Rectangle (210,10 428x30), "Измеряемые параметры ИБП 2.2"
    Rectangle (30,80 200x30), "Фазные напряжения:"
    Rectangle (60,120 150x30), "Ua = %3.2f", text variable: PLC_PRG.module_in1_u1
    Rectangle (60,160 150x30), "Ub = %3.2f", text variable: PLC_PRG.module_in1_u2
    Rectangle (60,200 150x30), "Uc = %3.2f", text variable: PLC_PRG.module_in1_u3
    Rectangle (290,80 200x30), "Линейные напряжения:"
    Rectangle (320,120 150x30), "Uab = %3.2f", text variable: PLC_PRG.module_in1_Uab
    Rectangle (320,160 150x30), "Ubc = %3.2f", text variable: PLC_PRG.module_in1_Ubc
    Rectangle (320,200 150x30), "Uca = %3.2f", text variable: PLC_PRG.module_in1_Uca
    Rectangle (560,80 200x30), "Фазные токи:"
    Rectangle (590,120 150x30), "Ia = %3.2f", text variable: PLC_PRG.module_in2_Ia
    Rectangle (590,160 150x30), "Ib = %3.2f", text variable: PLC_PRG.module_in2_Ib
    Rectangle (590,200 150x30), "Ic = %3.2f", text variable: PLC_PRG.module_in2_Ic
    Rectangle (300,260 200x30), "Частота:"
    Rectangle (330,310 150x30), "f = %3.2f", text variable: PLC_PRG.module_in2_F
    Image (10,390 130x78), image: ImagePool.zit
    Image (660,390 130x76), image: ImagePool.entel
END_VISUALIZATION

// Device/Application/scheme
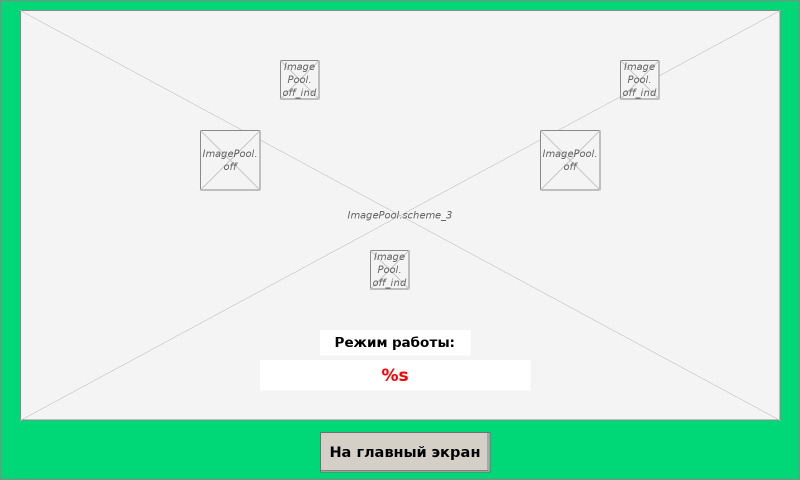
VISUALIZATION scheme  // 800x480
    Image (20,10 760x410), image: ImagePool.scheme_3
    Button (320,432 170x40), "На главный экран"
        OnMouseClick:  Assign=Visualization, Type=Assignment
    Image (620,60 39x39), image: ImagePool.off_ind
        p84334746: PLC_PRG.mv110_in_2
    Image (280,60 39x39), image: ImagePool.off_ind
        p84334746: PLC_PRG.mv110_in_1
    Image (370,250 39x39), image: ImagePool.off_ind
        p84334746: PLC_PRG.mv110_in_3
    Image (540,130 60x60), image: ImagePool.off
        p84334746: PLC_PRG.mv110_in_11
    Image (200,130 60x60), image: ImagePool.off
        p84334746: PLC_PRG.mv110_in_10
    Rectangle (320,330 150x25), "Режим работы:"
    Rectangle (260,360 270x30), "%s", text variable: PLC_PRG.mode
END_VISUALIZATION

(* text list AlarmGroup (id | default)
  44 | Отсутствует напряжение на секции
  43 | Отсутствует напряжение на вводе №2
  42 | Отсутствует напряжение на вводе №1
  41 | Пониженное напряжение  на секции №2 Uc = TRIGGERVALUE
  40 | Повышенное напряжение  на секции №2 Uc = TRIGGERVALUE
  39 | Пониженное напряжение на секции №2 Ub = TRIGGERVALUE
  38 | Повышенное напряжение  на секции №2 Ub = TRIGGERVALUE
  37 | Пониженное напряжение на секции №2 Ua = TRIGGERVALUE
  36 | Повышенное напряжение на секции №2 Ua = TRIGGERVALUE
  35 | Пониженное напряжение на секции №1 Uc = TRIGGERVALUE
  34 | Повышенное напряжение на секции №1 Uc = TRIGGERVALUE
  33 | Пониженное напряжение на секции №1 Ub = TRIGGERVALUE
  32 | Повышенное напряжение на секции №1 Ub = TRIGGERVALUE
  31 | Пониженное напряжени на секции №1 Ua = TRIGGERVALUE
  30 | Повышенное напряжение на секции №1 Ua = TRIGGERVALUE
  29 | Перегрузка Ic на секции шин
  28 | Перегрузка Ib на секции шин
  27 | Перегрузка Ia  на секции шин
  26 | Перегрузка Ic на вводе №2
  25 | Перегрузка Ib на вводе №2
  24 | Перегрузка Ia на вводе №2
  23 | Пониженное напряжение на вводе №2 Uc = TRIGGERVALUE
  22 | Повышенное напряжение на вводе №2 Uc = TRIGGERVALUE
  21 | Пониженное напряжение на вводе №2 Ub = TRIGGERVALUE
  20 | Повышенное напряжение на вводе №2 Ub = TRIGGERVALUE 
  19 | Пониженное напряжение  на вводе №2 Ua = TRIGGERVALUE
  18 | Повышенное напряжение  на вводе №2 Ua = TRIGGERVALUE
  17 | Перегрузка Ic на вводе №1
  16 | Перегрузка Ib на вводе №1
  15 | Перегрузка Ia на вводе №1
  14 | Пониженное напряжение Uc на вводе №1 = TRIGGERVALUE
  13 | Повышенное напряжение на вводе №1 Uc = TRIGGERVALUE
  12 | Пониженное напряжение на вводе №1 Ub = TRIGGERVALUE
  11 | Повышенное напряжение на вводе №1 Ub = TRIGGERVALUE
  10 | Пониженное напряжение  на вводе №1 Ua = TRIGGERVALUE
  9 | Повышенное напряжение  на вводе №1 Ua = TRIGGERVALUE
  8 | Авария ввода №2
  7 | Авария ввода №1
  6 | Авария секционного автомата
  5 | Пониженное напряжение
  4 | Ошибка_2
  3 | Ошибка_1
  2 | Предупреждение_3
  1 | Предупреждение_2
  0 | Предупреждение_1
   |  *)
